{attribute 'qualified_only'}
VAR_GLOBAL
	dm260 	: TcoCognexVision.TcoDatamanIO_v_5_x_x;
	dm8700 	: TcoCognexVision.TcoDatamanIO_v_5_x_x;
END_VAR

(* stored: Version 1.1.0.1, ProductVersion 3.1.4024.11
   GVL IO: Id {d37be50e-c2b3-0888-2f29-ec0e6f116694} *)
